Fanuc KAREL source: CNC_DYN_DISB.kl

PROGRAM T
%NOLOCKGROUP
VAR
 v0 : BOOLEAN
 v1 : STRING[40]
 v2 : INTEGER
BEGIN
 CNC_DYN_DISB(v0, v1, v2)
END T
